(* PLC project CodesysTest.project, PN2IC PLCopen CODESYS V3.5 SP17 Patch 3 *)
(* stored: creationDateTime 2022-06-20T21:06:04, modificationDateTime 2022-06-20T21:06:04 *)

PROGRAM flow\_2

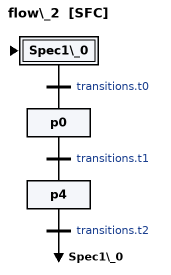
INITIAL_STEP Spec1\_0:
END_STEP
TRANSITION FROM Spec1\_0 TO p0
  := transitions.t0;
END_TRANSITION
STEP p0:
END_STEP
TRANSITION FROM p0 TO p4
  := transitions.t1;
END_TRANSITION
STEP p4:
END_STEP
TRANSITION FROM p4 TO Spec1\_0
  := transitions.t2;
END_TRANSITION
END_PROGRAM

PROGRAM flow\_1

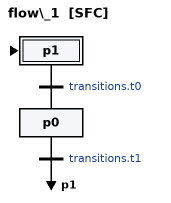
INITIAL_STEP p1:
END_STEP
TRANSITION FROM p1 TO p0
  := transitions.t0;
END_TRANSITION
STEP p0:
END_STEP
TRANSITION FROM p0 TO p1
  := transitions.t1;
END_TRANSITION
END_PROGRAM

PROGRAM Spec1

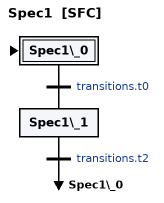
INITIAL_STEP Spec1\_0:
END_STEP
TRANSITION FROM Spec1\_0 TO Spec1\_1
  := transitions.t0;
END_TRANSITION
STEP Spec1\_1:
END_STEP
TRANSITION FROM Spec1\_1 TO Spec1\_0
  := transitions.t2;
END_TRANSITION
END_PROGRAM

PROGRAM flow\_4

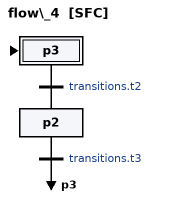
INITIAL_STEP p3:
END_STEP
TRANSITION FROM p3 TO p2
  := transitions.t2;
END_TRANSITION
STEP p2:
END_STEP
TRANSITION FROM p2 TO p3
  := transitions.t3;
END_TRANSITION
END_PROGRAM

PROGRAM transitions

 
END_PROGRAM

CONFIGURATION Application
  RESOURCE Application ON PLC
    VAR_GLOBAL  (* GVL *)
      t1 : BOOL;
      t2 : BOOL;
      t3 : BOOL;
      t0 : BOOL;
    END_VAR
    TASK MainTask(INTERVAL := T#20ms, PRIORITY := 1);
    PROGRAM flow\_2 WITH MainTask : flow\_2;
    PROGRAM flow\_1 WITH MainTask : flow\_1;
    PROGRAM Spec1 WITH MainTask : Spec1;
    PROGRAM flow\_4 WITH MainTask : flow\_4;
  END_RESOURCE
END_CONFIGURATION
